{attribute addProperty BoxType "EL6201-0000-0017"}
{attribute addProperty Id "Slave_4A_DI0BIT10.12525Slave_4A_DI1BIT10.12526Slave_4A_DI2BIT10.12527Slave_4A_DI3BIT10.12528Slave_4B_DI0BIT10.12529Slave_4B_DI1BIT10.12530Slave_4B_DI2BIT10.12531Slave_4B_DI3BIT10.12532"}
{attribute addProperty CRC "3407581132"}
{attribute addProperty SizeInBites "8"}
{attribute addProperty SizeInBytes "1"}
TYPE Slave_4_Inputs_CB1B8FCC :
STRUCT
	{attribute addProperty Name "Slave_4A_DI0"}
	Slave_4A_DI0 : BIT;
	{attribute addProperty Name "Slave_4A_DI1"}
	Slave_4A_DI1 : BIT;
	{attribute addProperty Name "Slave_4A_DI2"}
	Slave_4A_DI2 : BIT;
	{attribute addProperty Name "Slave_4A_DI3"}
	Slave_4A_DI3 : BIT;
	{attribute addProperty Name "Slave_4B_DI0"}
	Slave_4B_DI0 : BIT;
	{attribute addProperty Name "Slave_4B_DI1"}
	Slave_4B_DI1 : BIT;
	{attribute addProperty Name "Slave_4B_DI2"}
	Slave_4B_DI2 : BIT;
	{attribute addProperty Name "Slave_4B_DI3"}
	Slave_4B_DI3 : BIT;
END_STRUCT
END_TYPE

(* stored: Version 1.2.0.0, ProductVersion 3.1.4024.9
   DUT Slave_4_Inputs_CB1B8FCC: Id {ba32e7bd-80fe-4c6d-9c8c-88637b6d6bf1} *)
